(* PLC project Tc2_Utilities.FB_GetLocalAmsNetId Demo, tc3-libraries-kb TwinCAT 3.1 *)
(* stored: creationDateTime 2026-05-10T20:00:00, modificationDateTime 2026-05-10T20:00:00 *)

PROGRAM P_Demo_FB_GetLocalAmsNetId
  VAR
    fbFB_GetLocalAmsNetId : FB_GetLocalAmsNetId;  (* Tc2_Utilities.FB_GetLocalAmsNetId 实例 *)
    arg_bExecute : BOOL;  (* VAR_INPUT bExecute *)
    arg_tTimeOut : TIME;  (* VAR_INPUT tTimeOut *)
    out_bBusy : BOOL;  (* VAR_OUTPUT bBusy *)
    out_bError : BOOL;  (* VAR_OUTPUT bError *)
    out_nErrId : UDINT;  (* VAR_OUTPUT nErrId *)
    out_AddrString : T_AmsNetId;  (* VAR_OUTPUT AddrString *)
    out_AddrBytes : T_AmsNetIdArr;  (* VAR_OUTPUT AddrBytes *)
  END_VAR

            // ============================================================
// Tc2_Utilities.FB_GetLocalAmsNetId 演示程序（FB 实例）
// ============================================================
// 验证步骤：
//   1. 引用 Tc2_Utilities（及依赖类型所在库 Tc2_System 等）
//   2. 编译 + 登录
//   3. 按 doc.md 给 arg_* 赋值
//   4. 在线监视 out_* / io_* 输出
// ============================================================

fbFB_GetLocalAmsNetId(
    bExecute := arg_bExecute,
    tTimeOut := arg_tTimeOut,
    bBusy => out_bBusy,
    bError => out_bError,
    nErrId => out_nErrId,
    AddrString => out_AddrString,
    AddrBytes => out_AddrBytes
);

          
END_PROGRAM
